// TIA Portal V16 export
// export: Created 2021-07-12T14:47:14.1797967Z, ExportSetting WithDefaults, DisplayName Totally Integrated Automation Portal, DisplayVersion V16, DisplayName TIA Portal Version Control Interface, DisplayVersion V16, DisplayName TIA Portal Openness, DisplayVersion V16, DisplayName STEP 7 Professional, DisplayVersion V16, DisplayName STEP 7 Safety, DisplayVersion V16, DisplayName WinCC Professional, DisplayVersion V16
FUNCTION "Scale" : Void   // FC1, LAD
{ S7_Optimized_Access := 'TRUE' }
VERSION : 0.1
// stored: AutoNumber true, IsIECCheckEnabled false, SetENOAutomatically false, UDAEnableTagReadback false
   VAR_OUTPUT
      Scale_Out : Real;
   END_VAR
   VAR_TEMP
      AUX : Real;
   END_VAR
BEGIN

REGION Network 1
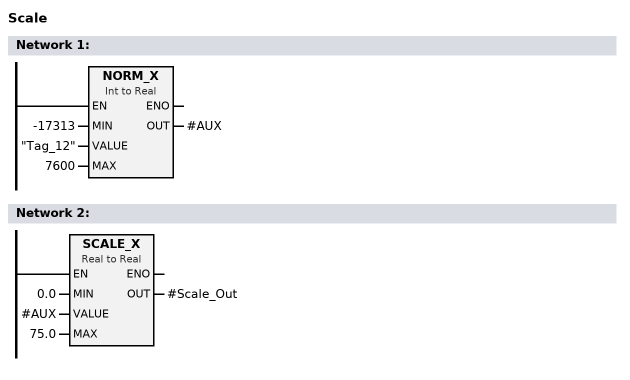
   RUNG wire#powerrail
      { S7_Templates := "[SrcType := Int, DestType := Real]" } Normalize(min := -17313, value := "Tag_12", max := 7600, out => #AUX)
   END_RUNG
   // the same network as SCL:
   #AUX := NORM_X(MIN := -17313, VALUE := "Tag_12", MAX := 7600);
END_REGION

REGION Network 2
   RUNG wire#powerrail
      { S7_Templates := "[SrcType := Real, DestType := Real]" } Scale(min := 0.0, value := #AUX, max := 75.0, out => #Scale_Out)
   END_RUNG
   // the same network as SCL:
   #Scale_Out := SCALE_X(MIN := 0.0, VALUE := #AUX, MAX := 75.0);
END_REGION
END_FUNCTION
